Omron CX-Programmer project NewProject (CX-Programmer 9.73)

# PLC NewPLC1: CP2E-N N

## Global symbols (name address type ; comment)
0.00 BOOL  ; Ax0 Org Sensor
0.01 BOOL  ; Ax0 CW-Limit
0.02 BOOL  ; Ax0 CCW-Limit
0.11 BOOL  ; EMG/PB
100.04 BOOL  ; Q_Break1
100.05 BOOL  ; Q_Break2
100.06 BOOL  ; Q_EN1
100.07 BOOL  ; Q_EN2
101.07 BOOL  ; Test Break
280.07 BOOL  ; Ax0 Error
A276 CHANNEL  ; Ax0 Current PLS
A277 CHANNEL  ; Ax1 Current PLS
A278 CHANNEL  ; Point B Data
A280.04 BOOL  ; Ax0 Busy
A280.05 BOOL  ; Ax0 No Org
A280.06 BOOL  ; Ax0 at Org
A280.07 BOOL  ; Ax0 Error
A281.04 BOOL  ; Ax1 Bussy
A540.08 BOOL  ; Ax0 CW-Limit Input
A540.09 BOOL  ; Ax0 CCW-Limit Input
D0 CHANNEL  ; $?St$Bk?_#[220] / Value"0"$?St$Bk?_#[220]
D10 CHANNEL  ; Point A Data
D100 CHANNEL  ; Axo Acceleration
D101 CHANNEL  ; Ax0 Deceleration
D102 CHANNEL  ; Target Frequency
D104 CHANNEL  ; Ax0 Number PLS Output
D105 CHANNEL  ; Ax1 Number PLS Output
D106 CHANNEL  ; Start Frequency
D110 CHANNEL  ; Ax1 Acceleration
D111 CHANNEL  ; Ax1 Deceleration
D112 CHANNEL  ; Target Frequency1
D114 CHANNEL  ; Ax1 Number PLS Output
D116 CHANNEL  ; Start Frequncy1
D12 CHANNEL  ; Point B Data
D14 CHANNEL  ; Point C Data
D20 CHANNEL  ; Point2 A Data
D22 CHANNEL  ; Point2 B Data
D24 CHANNEL  ; Point2 C Data
D276 CHANNEL  ; Ax0 Current PLS
D277 CHANNEL  ; Ax1 Current PLS
T010 BOOL  ; Ax0 Jog High
T011 BOOL  ; Ax1 Jog High
W0.02 BOOL  ; PB Ax0 Org
W0.03 BOOL  ; Axis0 Jog(+)
W0.04 BOOL  ; Axis Jog(-)
W0.05 BOOL  ; PB Ax1 Org
W0.06 BOOL  ; Axis1 Jog(+)
W0.07 BOOL  ; Axis1 Jog(-)
W100.00 BOOL  ; No Use
W100.01 BOOL  ; BREAK ACTIVE
W100.02 BOOL  ; ENA 1
W100.03 BOOL  ; INI MOTOR
W100.04 BOOL  ; BREAK 2
W100.07 BOOL  ; ENA 2
W10.00 BOOL  ; Ax0 Recover Org Start
W10.01 BOOL  ; Ax0 Recover Org Start PLS
W10.02 BOOL  ; Ax0 Org Return
W10.03 BOOL  ; Ax0 Org Returning
W10.04 BOOL  ; Ax0 at Org
W10.05 BOOL  ; Init
W10.06 BOOL  ; Ax0 Moving
W10.10 BOOL  ; Ax1 Recover Org Start
W10.14 BOOL  ; Ax1 Recover
W10.15 BOOL  ; Ax0 Recover C
W11.00 BOOL  ; 10.01
W11.01 BOOL  ; Ax1 Recover Org Start PLS
W11.10 BOOL  ; Teach2 Point A
W11.11 BOOL  ; Teach2 Point B
W11.12 BOOL  ; Teach2 Point C
W1.00 BOOL  ; Ax0 Jog High Speed
W1.01 BOOL  ; Ax0 Jog(+)
W1.02 BOOL  ; Ax0 Jog(-)
W1.03 BOOL  ; Ax1 Jog High Speed
W1.04 BOOL  ; Ax1 Jog(+)
W1.05 BOOL  ; Ax1 Jog(-)
W1.10 BOOL  ; Teach Point A
W1.11 BOOL  ; Teah Point B
W1.12 BOOL  ; Teach Point C
W20.00 BOOL  ; No Use
W20.01 BOOL  ; Sens Home
W20.02 BOOL  ; Sens CW
W20.03 BOOL  ; Sens CCW
W22.00 BOOL  ; Point2 A Run
W23.00 BOOL  ; Point2 A Proses
W23.02 BOOL  ; Ax1 at Point A
W2.00 BOOL  ; Point A Run
W2.01 BOOL  ; Point B Run
W2.02 BOOL  ; Point C Run
W32.02 BOOL  ; Ax1 at Point A
W3.00 BOOL  ; Point A Proses
W3.01 BOOL  ; Point A Trigger
W3.02 BOOL  ; Ax0 at Point A
W4.00 BOOL  ; Point B Process
W4.01 BOOL  ; Point B Trigger
W4.02 BOOL  ; Ax0 at Point B
W5.00 BOOL  ; Point C Progress
W5.01 BOOL  ; Point C Trigger
W5.02 BOOL  ; Ax0 at Point C
W99.01 BOOL  ; LOCK

## Program NewProgram1 (cyclic task 0)

### Section Axis0_Org

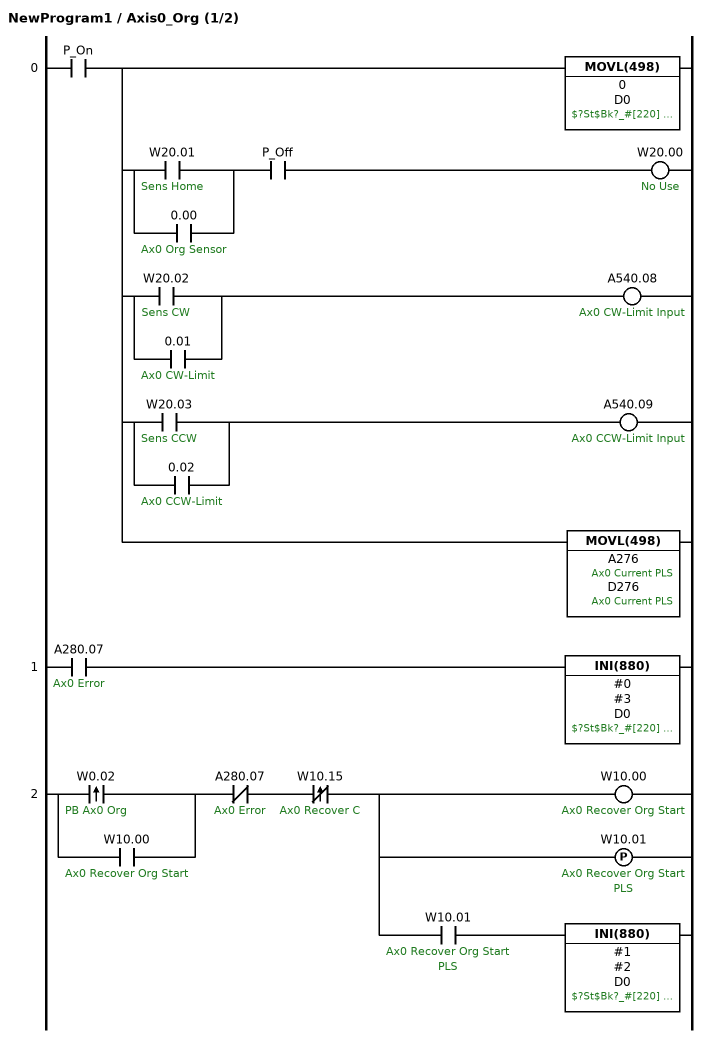
; rung 0
LD P_On
OUT TR0
MOVL(498) 0 D0  ; $?St$Bk?_#[220] / Value"0"$?St$Bk?_#[220]
LD W20.01  ; Sens Home
OR 0.00  ; Ax0 Org Sensor
ANDLD
AND P_Off
OUT W20.00  ; No Use
LD TR0
LD W20.02  ; Sens CW
OR 0.01  ; Ax0 CW-Limit
ANDLD
OUT A540.08  ; Ax0 CW-Limit Input
LD TR0
LD W20.03  ; Sens CCW
OR 0.02  ; Ax0 CCW-Limit
ANDLD
OUT A540.09  ; Ax0 CCW-Limit Input
LD TR0
MOVL(498) A276 D276  ; Ax0 Current PLS
; rung 1
LD A280.07  ; Ax0 Error
INI(880) #0 #3 D0  ; $?St$Bk?_#[220] / Value"0"$?St$Bk?_#[220]
; rung 2
@LD W0.02  ; PB Ax0 Org
OR W10.00  ; Ax0 Recover Org Start
ANDNOT A280.07  ; Ax0 Error
@ANDNOT W10.15  ; Ax0 Recover C
OUT W10.00  ; Ax0 Recover Org Start
DIFU(013) W10.01  ; Ax0 Recover Org Start PLS
AND W10.01  ; Ax0 Recover Org Start PLS
INI(880) #1 #2 D0  ; $?St$Bk?_#[220] / Value"0"$?St$Bk?_#[220]

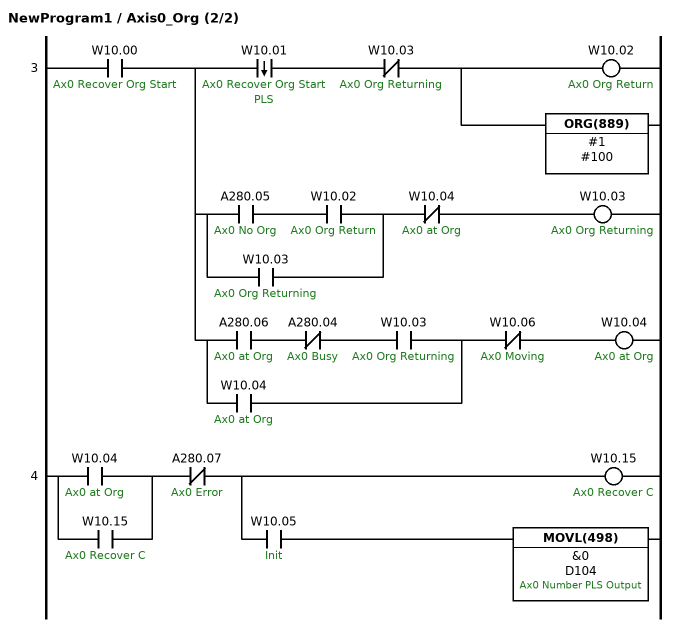
; rung 3
LD W10.00  ; Ax0 Recover Org Start
OUT TR0
%AND W10.01  ; Ax0 Recover Org Start PLS
ANDNOT W10.03  ; Ax0 Org Returning
OUT W10.02  ; Ax0 Org Return
ORG(889) #1 #100
LD TR0
LD A280.05  ; Ax0 No Org
AND W10.02  ; Ax0 Org Return
OR W10.03  ; Ax0 Org Returning
ANDLD
ANDNOT W10.04  ; Ax0 at Org
OUT W10.03  ; Ax0 Org Returning
LD TR0
LD A280.06  ; Ax0 at Org
ANDNOT A280.04  ; Ax0 Busy
AND W10.03  ; Ax0 Org Returning
OR W10.04  ; Ax0 at Org
ANDLD
ANDNOT W10.06  ; Ax0 Moving
OUT W10.04  ; Ax0 at Org
; rung 4
LD W10.04  ; Ax0 at Org
OR W10.15  ; Ax0 Recover C
ANDNOT A280.07  ; Ax0 Error
OUT W10.15  ; Ax0 Recover C
AND W10.05  ; Init
MOVL(498) &0 D104  ; Ax0 Number PLS Output

### Section Axis0_Jog

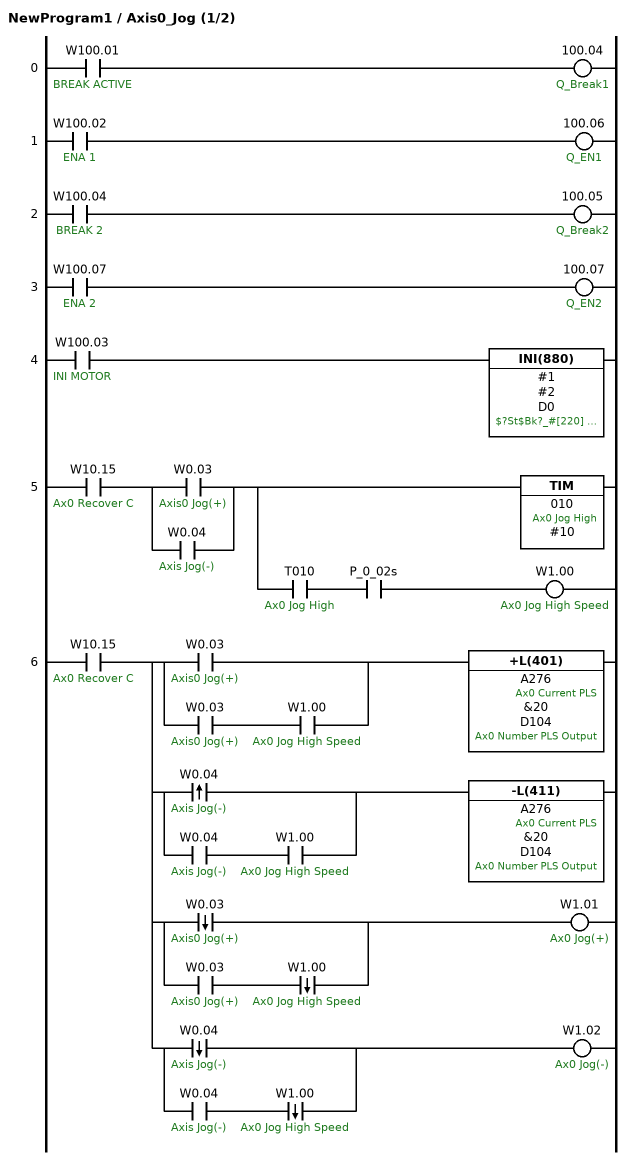
; rung 0
LD W100.01  ; BREAK ACTIVE
OUT 100.04  ; Q_Break1
; rung 1
LD W100.02  ; ENA 1
OUT 100.06  ; Q_EN1
; rung 2
LD W100.04  ; BREAK 2
OUT 100.05  ; Q_Break2
; rung 3
LD W100.07  ; ENA 2
OUT 100.07  ; Q_EN2
; rung 4
LD W100.03  ; INI MOTOR
INI(880) #1 #2 D0  ; $?St$Bk?_#[220] / Value"0"$?St$Bk?_#[220]
; rung 5
LD W10.15  ; Ax0 Recover C
LD W0.03  ; Axis0 Jog(+)
OR W0.04  ; Axis Jog(-)
ANDLD
TIM 010 #10  ; Ax0 Jog High
AND T010  ; Ax0 Jog High
AND P_0_02s
OUT W1.00  ; Ax0 Jog High Speed
; rung 6
LD W10.15  ; Ax0 Recover C
OUT TR0
LD W0.03  ; Axis0 Jog(+)
LD W0.03  ; Axis0 Jog(+)
AND W1.00  ; Ax0 Jog High Speed
ORLD
ANDLD
+L(401) A276 &20 D104  ; Ax0 Current PLS, Ax0 Number PLS Output
LD TR0
@LD W0.04  ; Axis Jog(-)
LD W0.04  ; Axis Jog(-)
AND W1.00  ; Ax0 Jog High Speed
ORLD
ANDLD
-L(411) A276 &20 D104  ; Ax0 Current PLS, Ax0 Number PLS Output
LD TR0
%LD W0.03  ; Axis0 Jog(+)
LD W0.03  ; Axis0 Jog(+)
%AND W1.00  ; Ax0 Jog High Speed
ORLD
ANDLD
OUT W1.01  ; Ax0 Jog(+)
LD TR0
%LD W0.04  ; Axis Jog(-)
LD W0.04  ; Axis Jog(-)
%AND W1.00  ; Ax0 Jog High Speed
ORLD
ANDLD
OUT W1.02  ; Ax0 Jog(-)

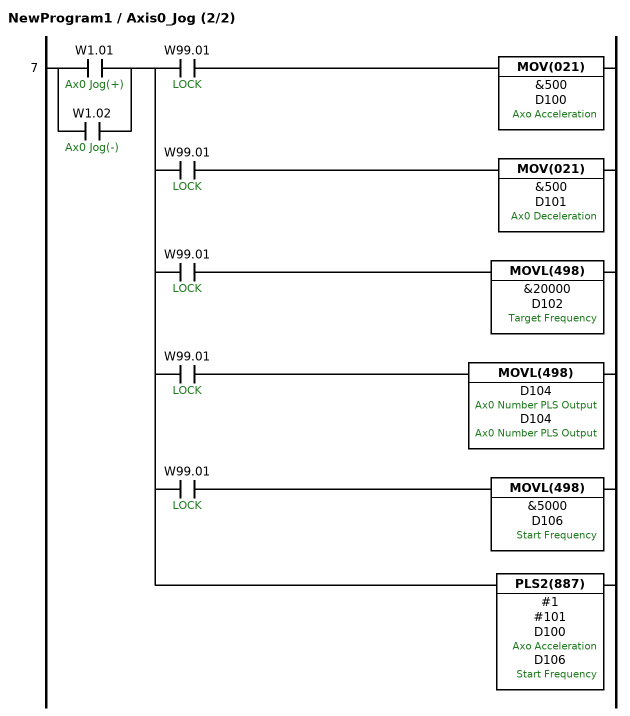
; rung 7
LD W1.01  ; Ax0 Jog(+)
OR W1.02  ; Ax0 Jog(-)
OUT TR0
AND W99.01  ; LOCK
MOV(021) &500 D100  ; Axo Acceleration
LD TR0
AND W99.01  ; LOCK
MOV(021) &500 D101  ; Ax0 Deceleration
LD TR0
AND W99.01  ; LOCK
MOVL(498) &20000 D102  ; Target Frequency
LD TR0
AND W99.01  ; LOCK
MOVL(498) D104 D104  ; Ax0 Number PLS Output
LD TR0
AND W99.01  ; LOCK
MOVL(498) &5000 D106  ; Start Frequency
LD TR0
PLS2(887) #1 #101 D100 D106  ; Axo Acceleration, Start Frequency

### Section Axis0_Point_Run

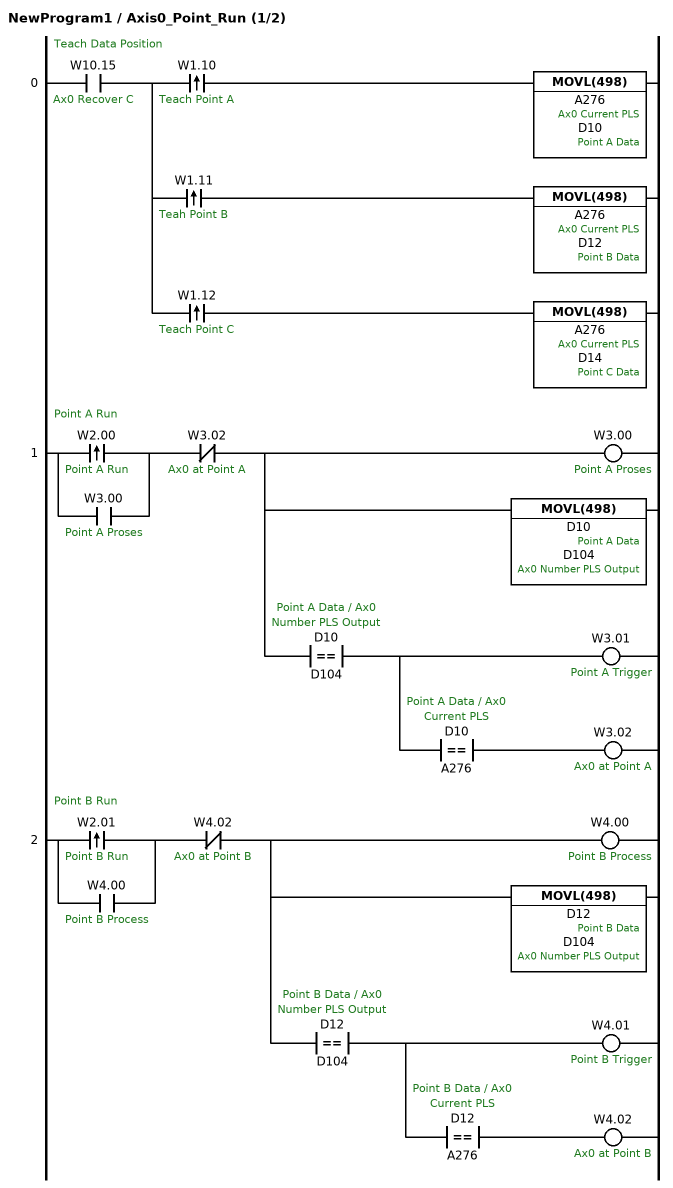
; rung 0: Teach Data Position
LD W10.15  ; Ax0 Recover C
OUT TR0
@AND W1.10  ; Teach Point A
MOVL(498) A276 D10  ; Ax0 Current PLS, Point A Data
LD TR0
@AND W1.11  ; Teah Point B
MOVL(498) A276 D12  ; Ax0 Current PLS, Point B Data
LD TR0
@AND W1.12  ; Teach Point C
MOVL(498) A276 D14  ; Ax0 Current PLS, Point C Data
; rung 1: Point A Run
@LD W2.00  ; Point A Run
OR W3.00  ; Point A Proses
ANDNOT W3.02  ; Ax0 at Point A
OUT W3.00  ; Point A Proses
MOVL(498) D10 D104  ; Point A Data, Ax0 Number PLS Output
AND=L(301) D10 D104  ; Point A Data, Ax0 Number PLS Output
OUT W3.01  ; Point A Trigger
AND=L(301) D10 A276  ; Point A Data, Ax0 Current PLS
OUT W3.02  ; Ax0 at Point A
; rung 2: Point B Run
@LD W2.01  ; Point B Run
OR W4.00  ; Point B Process
ANDNOT W4.02  ; Ax0 at Point B
OUT W4.00  ; Point B Process
MOVL(498) D12 D104  ; Point B Data, Ax0 Number PLS Output
AND=L(301) D12 D104  ; Point B Data, Ax0 Number PLS Output
OUT W4.01  ; Point B Trigger
AND=L(301) D12 A276  ; Point B Data, Ax0 Current PLS
OUT W4.02  ; Ax0 at Point B

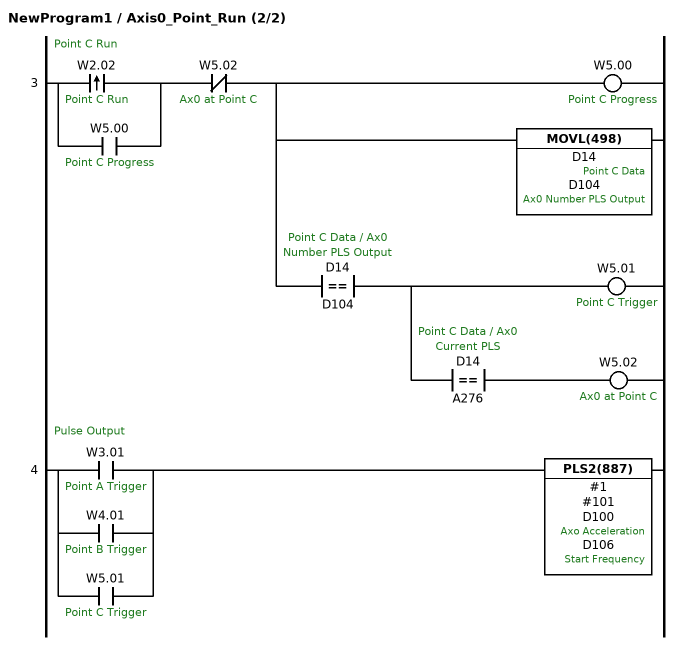
; rung 3: Point C Run
@LD W2.02  ; Point C Run
OR W5.00  ; Point C Progress
ANDNOT W5.02  ; Ax0 at Point C
OUT W5.00  ; Point C Progress
MOVL(498) D14 D104  ; Point C Data, Ax0 Number PLS Output
AND=L(301) D14 D104  ; Point C Data, Ax0 Number PLS Output
OUT W5.01  ; Point C Trigger
AND=L(301) D14 A276  ; Point C Data, Ax0 Current PLS
OUT W5.02  ; Ax0 at Point C
; rung 4: Pulse Output
LD W3.01  ; Point A Trigger
OR W4.01  ; Point B Trigger
OR W5.01  ; Point C Trigger
PLS2(887) #1 #101 D100 D106  ; Axo Acceleration, Start Frequency

### Section END
; rung 0
END(001)